	IF CommonTypesAndFunctions.StrEqualsAtStartWithDelimiter(str1:= ADR(LastTreeName), str2:= Data.PayloadString, delimiter:= SplitPayloadChar) THEN
		//now search split char
		StrPt := Data.PayloadString;
		StrPt := StrPt + TO_DWORD(CommonTypesAndFunctions.find(str1 := StrPt, str2:= ADR(SplitPayloadChar))) + 1;
		Target := StrPt^;
	END_IF
END_IF
END_METHOD

METHOD initAsFindTopic : BOOL
VAR_INPUT
END_VAR
getLastTreeName();
splitPayload := FALSE;
splitTopic := TRUE;
END_METHOD

METHOD getLastTreeName : BOOL
VAR_INPUT
END_VAR
LastTreeName := CommonTypesAndFunctions.FindLastDot(ADR(instanceName))^;
END_METHOD

METHOD initAsFindPayload : BOOL
VAR_INPUT
	//only first char is selected
	splitChar:STRING;
END_VAR
getLastTreeName();
splitPayload := TRUE;
splitTopic := FALSE;

SplitPayloadChar := CommonTypesAndFunctions.GetChar(in:= splitChar);
END_METHOD

END_FUNCTION_BLOCK

// MQTT/TestCases/Test Interfaces/exampleForFbs
FUNCTION_BLOCK exampleForFbs
VAR_INPUT
END_VAR
VAR_OUTPUT
END_VAR
VAR
	//the MQTT client
	//client:ClientWrapper;
	//some reciving FBs
	FirstExtReceiver:FooBarReceivingFB;
	SecondExtReceiver:FooBarReceivingFB;
	ThirdExtReceiver:FooBarReceivingFB;
	FourthExtReceiver:FooBarReceivingFB;
	//a Array of receiving FBs
	ArrayReceive:ARRAY[0..9] OF FooBarReceivingFB;
	
	//the collector of the FBs
	stock:CallbackCollector;
END_VAR



(*
client(
	broker:= 'test.mosquitto.org:1883', 
	connect:= TRUE, 
	tls:= FALSE);

	*)

END_FUNCTION_BLOCK

// MQTT/Function Blocks/CallbackFBs/Callback Collector/ReceiveValueWithStrucur
FUNCTION_BLOCK ReceiveValueWithStrucur EXTENDS ReceiveValue
VAR_INPUT
END_VAR
VAR_OUTPUT
END_VAR
VAR
	InstanceName:CommonTypesAndFunctions.GetInstanceName;
	localCompString:STRING(255);
END_VAR

METHOD InitReceiveStructur : BOOL
VAR_INPUT
	
	TopicLevel:USINT;
	//this typ is my received string
	ValueTyp:CommonTypesAndFunctions.VAR_TYPES; 
	//if set to true and hit we will return true, else false...
	returnHit: BOOL;
END_VAR
VAR
	tString:STRING(255);
	cmpByte:BYTE;
	bytePointer:POINTER TO BYTE;
	StringPointer:POINTER TO STRING;
	i:UINT;
END_VAR

tString:= InstanceName.GetInstanceTopic();

cmpByte:= CommonTypesAndFunctions.GetChar('/');

bytePointer := ADR(tString) + CommonTypesAndFunctions.len(ADR(tString));

i := 0;

WHILE bytePointer >= ADR(tString) DO
	IF bytePointer^ = cmpByte THEN
		i := i + 1; 
	END_IF
	
	IF i = TopicLevel THEN
		
		StringPointer := bytePointer + 1;
		//ReceiveTopic := GVL_ZIGBEE.TextZigbeeTopic;
		//ReceiveTopic := CONCAT(STR1:= ReceiveTopic, STR2:= StringPointer^); 
		localCompString := StringPointer^;
		initAsFindTopic(compString:= ADR(localCompString), ValueTyp:= ValueTyp, returnHit:= returnHit);
		RETURN;
	END_IF
	bytePointer := bytePointer - 1;
END_WHILE
localCompString := tString;
initAsFindTopic(compString:= ADR(localCompString), ValueTyp:= ValueTyp, returnHit:= returnHit);
END_METHOD

END_FUNCTION_BLOCK

// MQTT/Function Blocks/CallbackFBs/Callback Collector/ReceiveValue
(*
Receives one value from a MQTT publish packet.
It can check diffrent sources to determinate if the data is for this Value....

*)
FUNCTION_BLOCK ReceiveValue IMPLEMENTS MQTT_SUBSCRIBE_CALLBACK
VAR_INPUT
END_VAR
VAR_OUTPUT
	//your desired payload...
	MQTTReceived:CommonTypesAndFunctions.ALL_TYPES_UNION;
END_VAR
VAR
	//pointer to target
	TargetPointer:CommonTypesAndFunctions.ALL_TYPES_UNION_POINTER;
	//Target var type
	MyValueTyp:CommonTypesAndFunctions.VAR_TYPES;
	//an this is the split char...
	SplitPayloadChar: BYTE;
	//compare with this...
	MyCompString:POINTER TO STRING;
	//and this for Payload
	MyCompStringPayload:POINTER TO STRING;
	//if set to true and hit we will return true, else false...
	MyReturnHit: BOOL;
	ReceiveType : RECEIVE_TYPS;
END_VAR


METHOD PublishReceived : BOOL
VAR_INPUT
	(*Collection of received Data*)
	Data	: CALLBACK_DATA;
END_VAR
VAR
	StrPt : POINTER TO STRING;
END_VAR
CASE ReceiveType OF
	RECEIVE_TYPS.FIND_LAST_TOPIC:	
		//now search the right topic 
		IF CommonTypesAndFunctions.StrEquals(str1:= Data.TopicOutSplit^.Topics[Data.TopicOutSplit^.ValidFields - 1], str2:= MyCompString) THEN
			CommonTypesAndFunctions.GetValueFromStringPt(TypeOfValue:= MyValueTyp ,Target:= TargetPointer, str:= DATA.PayloadString);
			PublishReceived := MyReturnHit;
		END_IF
	RECEIVE_TYPS.FIND_PAYLOAD:
		IF CommonTypesAndFunctions.StrEqualsAtStartWithDelimiter(str1:= MyCompString, str2:= Data.PayloadString, delimiter:= SplitPayloadChar) THEN
			//now search split char
			StrPt := Data.PayloadString;
			StrPt := StrPt + TO_DWORD(CommonTypesAndFunctions.find(str1 := StrPt, str2:= ADR(SplitPayloadChar))) + 1;
			CommonTypesAndFunctions.GetValueFromStringPt(TypeOfValue:= MyValueTyp ,Target:= TargetPointer, str:= StrPt);
			PublishReceived := MyReturnHit;
		END_IF
	RECEIVE_TYPS.FIND_LAST_TOPIC_AND_PAYLOAD:
		//now search the right topic and payload
		IF CommonTypesAndFunctions.StrEquals(str1:= Data.TopicOut, str2:= MyCompString) THEN
			IF CommonTypesAndFunctions.StrEqualsAtStartWithDelimiter(str1:= MyCompStringPayload, str2:= Data.PayloadString, delimiter:= SplitPayloadChar) THEN
				StrPt := Data.PayloadString;
				StrPt := StrPt + TO_DWORD(CommonTypesAndFunctions.find(str1 := StrPt, str2:= ADR(SplitPayloadChar))) + 1;
				CommonTypesAndFunctions.GetValueFromStringPt(TypeOfValue:= MyValueTyp ,Target:= TargetPointer, str:= StrPt);
				PublishReceived := MyReturnHit;
			END_IF
		END_IF
	RECEIVE_TYPS.FIND_TOPIC:
		//now search the right topic 
		IF CommonTypesAndFunctions.StrEquals(str1:= Data.TopicOut, str2:= MyCompString) THEN
			CommonTypesAndFunctions.GetValueFromStringPt(TypeOfValue:= MyValueTyp ,Target:= TargetPointer, str:= DATA.PayloadString);
			PublishReceived := MyReturnHit;
		END_IF
END_CASE
END_METHOD

METHOD initAsFindPayload : BOOL
VAR_INPUT
	//only first char is selected
	splitChar:STRING;
	//this i'm searching
	compString : POINTER TO STRING;
	//this typ is my received string
	ValueTyp:CommonTypesAndFunctions.VAR_TYPES; 
	//if set to true and hit we will return true, else false...
	returnHit: BOOL;
END_VAR
ReceiveType := RECEIVE_TYPS.FIND_PAYLOAD;

SplitPayloadChar := CommonTypesAndFunctions.GetChar(in:= splitChar);
MyCompString := compString;
MyValueTyp := ValueTyp;
makePointer();
MyReturnHit := returnHit;
END_METHOD

(*this will only check the lowest topic level*)
METHOD initAsFindTopic : BOOL
VAR_INPUT
	//this i'm searching
	compString : POINTER TO STRING;
	//this typ is my received string
	ValueTyp:CommonTypesAndFunctions.VAR_TYPES; 
	//if set to true and hit we will return true, else false...
	returnHit: BOOL;
END_VAR
ReceiveType := RECEIVE_TYPS.FIND_TOPIC;
MyCompString := compString;
MyValueTyp := ValueTyp;
makePointer();
MyReturnHit := returnHit;
END_METHOD

METHOD makePointer : BOOL
VAR_INPUT
END_VAR
TargetPointer := CommonTypesAndFunctions.MakeAllTypesPointer(fromWho:= adr(MQTTReceived), myType:= MyValueTyp);
END_METHOD

(*this will check the whole topic!*)
METHOD initAsFindTopicAndPayload : BOOL
VAR_INPUT
	//only first char is selected
	splitChar:STRING;
	//this topic i'm searching
	compStringTopic : POINTER TO STRING;
	//this payload i'm searching
	compStringPayload : POINTER TO STRING;
	//this typ is my received string
	ValueTyp:CommonTypesAndFunctions.VAR_TYPES; 
	//if set to true and hit we will return true, else false...
	returnHit: BOOL;
END_VAR
ReceiveType := RECEIVE_TYPS.FIND_LAST_TOPIC_AND_PAYLOAD;
SplitPayloadChar := CommonTypesAndFunctions.GetChar(in:= splitChar);
MyCompString := compStringTopic;
MyCompStringPayload := compStringPayload;
MyValueTyp := ValueTyp;
makePointer();
MyReturnHit := returnHit;
END_METHOD

METHOD SetOutput : BOOL
VAR_INPUT
	value:CommonTypesAndFunctions.ALL_TYPES_UNION;
END_VAR
MQTTReceived := value;
END_METHOD

METHOD initAsFindLastTopic : BOOL
VAR_INPUT
	//this i'm searching
	compString : POINTER TO STRING;
	//this typ is my received string
	ValueTyp:CommonTypesAndFunctions.VAR_TYPES; 
	//if set to true and hit we will return true, else false...
	returnHit: BOOL;
END_VAR
ReceiveType := RECEIVE_TYPS.FIND_LAST_TOPIC;
MyCompString := compString;
MyValueTyp := ValueTyp;
makePointer();
MyReturnHit := returnHit;
END_METHOD

END_FUNCTION_BLOCK

// MQTT/Function Blocks/CallbackFBs/Callback Collector/ReceiveString
FUNCTION_BLOCK ReceiveString IMPLEMENTS MQTT_SUBSCRIBE_CALLBACK
VAR_INPUT
END_VAR
VAR_OUTPUT
	//your desired payload...
	MQTTReceived:STRING(255);
END_VAR
VAR
	//if set to true we search the instance name in the lowest topic
	splitTopic: BOOL;
	//if set to true we search the instance name in Payload separatet by the split char 
	splitPayload: BOOL;
	//an this is the split char...
	SplitPayloadChar: BYTE;
	//compare with this...
	MyCompString:POINTER TO STRING;
	//if set to true and hit we will return true, else false...
	MyReturnHit: BOOL;
END_VAR

METHOD PublishReceived : BOOL
VAR_INPUT
	(*Collection of received Data*)
	Data	: CALLBACK_DATA;
	
END_VAR
VAR
	StrPt : POINTER TO STRING(255);
END_VAR
// no we can check if the topic/payload matches to my compare string 

//now search the right topic 
IF splitTopic THEN
	
	IF CommonTypesAndFunctions.StrEquals(str1:= Data.TopicOut, str2:= MyCompString) THEN
		StrPt := Data.PayloadString;
		MQTTReceived := StrPt^;
		PublishReceived := MyReturnHit;
	END_IF

END_IF

//now look into the payload
IF splitPayload THEN
	
	IF CommonTypesAndFunctions.StrEqualsAtStartWithDelimiter(str1:= MyCompString, str2:= Data.PayloadString, delimiter:= SplitPayloadChar) THEN
		//now search split char
		StrPt := Data.PayloadString;
		StrPt := StrPt + TO_DWORD(CommonTypesAndFunctions.find(str1 := StrPt, str2:= ADR(SplitPayloadChar))) + 1;
		MQTTReceived := StrPt^;
		PublishReceived := MyReturnHit;
	END_IF
END_IF
END_METHOD

METHOD initAsFindTopic : BOOL
VAR_INPUT
	//this i'm searching
	compString : POINTER TO STRING;
	//if set to true and hit we will return true, else false...
	returnHit: BOOL;
END_VAR

splitPayload := FALSE;
splitTopic := TRUE;
MyCompString := compString;
MyReturnHit := returnHit;
END_METHOD

METHOD initAsFindPayload : BOOL
VAR_INPUT
	//only first char is selected
	splitChar:STRING;
	//this i'm searching
	compString : POINTER TO STRING;
	//if set to true and hit we will return true, else false...
	returnHit: BOOL;
END_VAR

splitPayload := TRUE;
splitTopic := FALSE;

SplitPayloadChar := CommonTypesAndFunctions.GetChar(in:= splitChar);
MyCompString := compString;
MyReturnHit := returnHit;
END_METHOD

END_FUNCTION_BLOCK

// MQTT/TestCases/TestLongPublish
FUNCTION_BLOCK TestLongPublish
VAR_INPUT
	broker:STRING := 'test.mosquitto.org:1883';
END_VAR
VAR_OUTPUT
END_VAR
VAR
	longPayload:STRING(8000):='';
	longTopic:STRING(8000):=('TestTopic/');
	longPayloadReceive:STRING(8000);
	longTopicReceive:STRING(8000);
	init: BOOL;
	i1:UINT;
	i2:UINT;
	countAsciis :UINT := 48;
	pt1:POINTER TO BYTE;
	pt2:POINTER TO BYTE;
	
	step : UINT; 
	
	MQTT:HANDLE_MQTT;
	
	MQTT_IN_OUT:MQTT_IN_OUT;
	
	ComConfig:COM_CONFIG;
	
	pup:MQTTPublish;
	send: BOOL;

	
	SUB1:MQTTSubscribe;
	subscribe: BOOL;

	callback : SingelStringCallback;
	
	
	connect: BOOL;

	nextRung:ton;
	lenPayload:UINT;
	lenTopic:uint;
	
END_VAR

IF NOT init THEN
	init := TRUE;
	SUB1.SetMqttInOut(MQTT_IN_OUT := ADR(MQTT_IN_OUT));
	pup.SetMqttInOut(MQTT_IN_OUT := ADR(MQTT_IN_OUT));
	ComConfig.MaxPayloadSize := 20000;
	ComConfig.MaxTopicLevels := 10;
	ComConfig.MaxTopicElementSize := 10000;
	
	MQTT_IN_OUT.ClientID := 'TestCodesys';
	MQTT_IN_OUT.COM_CONFIG := ComConfig;
	//firs build some nice pacload ...
	pt1 := ADR(longPayload);
	pt2 := ADR(longTopic);
	pt2 := pt2 + 10;
	FOR i1 := 0 TO 8000 / countAsciis - 1 DO
		FOR i2 := 0 TO countAsciis - 1 DO
			pt1^ := TO_BYTE(i2 + 16#30); //16#30 --> ASCII zero
			pt2^ := TO_BYTE(i2 + 16#30); //16#30 --> ASCII zero
			pt1 := pt1 + 1;
			pt2 := pt2 + 1;
		END_FOR
	END_FOR
	//need termination...
	pt1^:= 0;
	pt2^:= 0;
	callback.Init(payload:= ADR(longPayloadReceive), topic:= ADR(longTopicReceive));
END_IF

SUB1(
	Subscribe:= subscribe, 
	Topic:= ADR('TestTopic/#'), 
	QoSSubscribe:= QoS.ExactlyOnce, 
	ExpectingString:= TRUE, 
	Callback:= callback);

	
	pup(
	Topic:= ADR(longTopic), 
	PayloadString:= ADR(longPayload), 
	PublishAsString:= TRUE, 
	QoSIn:= Qos.ExactlyOnce, 
	MRetain:= FALSE, 
	send:= send);

MQTT(
	MQTT_IN_OUT:= MQTT_IN_OUT, 
	ENABLE:= connect, 
	URL:= broker, 
	TIMEOUT:= T#5S);


CASE step OF 
	0://begin
		//connect
		connect := TRUE;
		step := 10;
	10://wait connected
		IF MQTT_IN_OUT.BROKER_CONNECTED THEN
			//subscribe
			subscribe := TRUE;		
			step := 20;
		END_IF
	20://wait subscribed
		IF SUB1.SubscribeDone THEN
			//send packet and check receive
			send := TRUE;
			step := 30;
		END_IF
		
	30:
		//reset send
		send := FALSE;
		step := 40;
	40:
		lenPayload:= CommonTypesAndFunctions.len(ADR(longPayloadReceive));
		lenTopic:= CommonTypesAndFunctions.len(ADR(longTopicReceive));
		//check if payload and topic received....
		IF CommonTypesAndFunctions.StrEquals(str1:= ADR(longPayload), str2:= ADR(longPayloadReceive)) AND
			CommonTypesAndFunctions.StrEquals(str1:= ADR(longTopic), str2:= ADR(longTopicReceive)) THEN
			//deled received strings
			longTopicReceive := '';
			longPayloadReceive := '';
			//go wait repeat
			step := 50;
		END_IF
		
	50:
		IF nextRung.Q THEN
			step := 0;
		END_IF
END_CASE

nextRung(IN:= step = 50, PT:= T#5S);

END_FUNCTION_BLOCK

// MQTT/TestCases/TestLongStringList
FUNCTION_BLOCK TestLongStringList
VAR_INPUT
	//use this input if you want to test with another broker
	client:STRING:='test.mosquitto.org:1883';//test.mosquitto.org
	
END_VAR
VAR_OUTPUT
END_VAR
VAR
	MQTTClient:HANDLE_MQTT;
	MQTT_IN_OUT:MQTT_IN_OUT;
	MQTTInfo:MQTT_INFO;
	publish:MQTTPublish;
	subscribe:MQTTSubscribe;
	ReceiveSubscribeTopic:STRING(255);
	
	ReceiveSubscribePayloadLong:STRING(500);
	State :MQTTState;
	init: BOOL;
	varSend: BOOL;
	timerSend:ton;
	t1:ton;
	t2:ton;
	Payload:STRING;
	//the method PublishReceved() is call when an publsih packet form the broker is received.
	StringCallback:ListStringCallback;
	//the array contains the targets and sub topics for receive
	CallBackTargets:ARRAY[0..1] OF LIST_STRING_CALLBACK_DATA := [(Target:=ADR(ReceiveSubscribePayloadLong), SubTopic:= ADR('Long'))];
	len1:UINT;
END_VAR

//here init is done
IF NOT init THEN
	init := TRUE;
	MQTT_IN_OUT.ClientID := CONCAT('CodesysMqtt',TO_STRING(TICKS.GetTick(xDummy:= TRUE)));
	//init state FB, so you only have to call state();without parameters... 
	State.Init(
	State:= ADR(t1.Q), 
	Topic:= ADR('CODESYS-MQTT-BY-SD/Long'), 
	StateName:= ADR(''), 
	StateValueOn:= ADR('LOOOOOOOOOOOOOOOOOOOOOOOOOOOOOOOOOOOOOOOOOOOOOOOOOOOOOOOOOOOOOOOOOOOOOOOOOOOOOOOOOOOOOOOOOOOOOOOOOOOOOOOOOOOOOOOOOOOOOOOOOOOOOOOOOOOOOOOOOOOOOOOOOOOOOOOOOOOOOOOOOOOOOOOOOOOOOOOOOOOOOOOOOOOOOOOOOOOOOOOOOOOOOOOOOOOOOOOOg:On'), 
	StateValueOff:= ADR('LOOOOOOOOOOOOOOOOOOOOOOOOOOOOOOOOOOOOOOOOOOOOOOOOOOOOOOOOOOOOOOOOOOOOOOOOOOOOOOOOOOOOOOOOOOOOOOOOOOOOOOOOOOOOOOOOOOOOOOOOOOOOOOOOOOOOOOOOOOOOOOOOOOOOOOOOOOOOOOOOOOOOOOOOOOOOOOOOOOOOOOOOOOOOOOOOOOOOOOOOOOOOOOOOOOOOOOOOg:Off'), 
	QoS:= QoS.ExactlyOnce, 
	RetainMqtt:= TRUE,
	MQTT_IN_OUT:= ADR(MQTT_IN_OUT));
	StringCallback.InitAsSplitTopic(ListData := ADR(CallBackTargets), LengthOfData:= 1);
	
	subscribe.SetMqttInOut(MQTT_IN_OUT:= ADR(MQTT_IN_OUT));
	
END_IF
//timer for repeating packets
t1(IN:= NOT t2.Q, PT:= T#1S, );
t2(IN:= t1.Q, PT:= T#1S);
//call of MQTT client
MQTTClient(
	MQTT_IN_OUT:= MQTT_IN_OUT, 
	ENABLE:= TRUE, 
	URL:= client, 
	TIMEOUT:= T#5S, 
	TLS:= FALSE);
//Subscribe to topic
subscribe(
	Subscribe:= TRUE, 
	Topic:= ADR('CODESYS-MQTT-BY-SD/#'), 
	QoSSubscribe:= QoS.ExactlyOnce, 
	ExpectingString:= TRUE,
	Callback:= StringCallback);
len1 := CommonTypesAndFunctions.len(str:= ADR(ReceiveSubscribePayloadLong));

//call of state FB
State();

END_FUNCTION_BLOCK

// MQTT/TestCases/TestStringPointer
FUNCTION_BLOCK TestStringPointer
VAR_INPUT
END_VAR
VAR_OUTPUT
END_VAR
VAR
	SFrom:STRING(2000):='ABCDEFGHIJKLMNOPQRSTUVWXYZABCDEFGHIJKLMNOPQRSTUVWXYZABCDEFGHIJKLMNOPQRSTUVWXYZABCDEFGHIJKLMNOPQRSTUVWXYZABCDEFGHIJKLMNOPQRSTUVWXYZABCDEFGHIJKLMNOPQRSTUVWXYZABCDEFGHIJKLMNOPQRSTUVWXYZABCDEFGHIJKLMNOPQRSTUVWXYZABCDEFGHIJKLMNOPQRSTUVWXYZABCDEFGHIJKLMNOPQRSTUVWXYZABCDEFGHIJKLMNOPQRSTUVWXYZABCDEFGHIJKLMNOPQRSTUVWXYZABCDEFGHIJKLMNOPQRSTUVWXYZABCDEFGHIJKLMNOPQRSTUVWXYZABCDEFGHIJKLMNOPQRSTUVWXYZABCDEFGHIJKLMNOPQRSTUVWXYZABCDEFGHIJKLMNOPQRSTUVWXYZABCDEFGHIJKLMNOPQRSTUVWXYZABCDEFGHIJKLMNOPQRSTUVWXYZABCDEFGHIJKLMNOPQRSTUVWXYZABCDEFGHIJKLMNOPQRSTUVWXYZABCDEFGHIJKLMNOPQRSTUVWXYZABCDEFGHIJKLMNOPQRSTUVWXYZABCDEFGHIJKLMNOPQRSTUVWXYZABCDEFGHIJKLMNOPQRSTUVWXYZABCDEFGHIJKLMNOPQRSTUVWXYZABCDEFGHIJKLMNOPQRSTUVWXYZABCDEFGHIJKLMNOPQRSTUVWXYZABCDEFGHIJKLMNOPQRSTUVWXYZABCDEFGHIJKLMNOPQRSTUVWXYZABCDEFGHIJKLMNOPQRSTUVWXYZABCDEFGHIJKLMNOPQRSTUVWXYZABCDEFGHIJKLMNOPQRSTUVWXYZABCDEFGHIJKLMNOPQRSTUVWXYZABCDEFGHIJKLMNOPQRSTUVWXYZABCDEFGHIJKLMNOPQRSTUVWXYZABCDEFGHIJKLMNOPQRSTUVWXYZABCDEFGHIJKLMNOPQRSTUVWXYZABCDEFGHIJKLMNOPQRSTUVWXYZABCDEFGHIJKLMNOPQRSTUVWXYZABCDEFGHIJKLMNOPQRSTUVWXYZABCDEFGHIJKLMNOPQRSTUVWXYZABCDEFGHIJKLMNOPQRSTUVWXYZABCDEFGHIJKLMNOPQRSTUVWXYZABCDEFGHIJKLMNOPQRSTUVWXYZABCDEFGHIJKLMNOPQRSTUVWXYZABCDEFGHIJKLMNOPQRSTUVWXYZABCDEFGHIJKLMNOPQRSTUVWXYZABCDEFGHIJKLMNOPQRSTUVWXYZABCDEFGHIJKLMNOPQRSTUVWXYZABCDEFGHIJKLMNOPQRSTUVWXYZABCDEFGHIJKLMNOPQRSTUVWXYZABCDEFGHIJKLMNOPQRSTUVWXYZABCDEFGHIJKLMNOPQRSTUVWXYZABCDEFGHIJKLMNOPQRSTUVWXYZABCDEFGHIJKLMNOPQRSTUVWXYZABCDEFGHIJKLMNOPQRSTUVWXYZABCDEFGHIJKLMNOPQRSTUVWXYZABCDEFGHIJKLMNOPQRSTUVWXYZABCDEFGHIJKLMNOPQRSTUVWXYZABCDEFGHIJKLMNOPQRSTUVWXYZABCDEFGHIJKLMNOPQRSTUVWXYZABCDEFGHIJKLMNOPQRSTUVWXYZABCDEFGHIJKLMNOPQRSTUVWXYZABCDEFGHIJKLMNOPQRSTUVWXYZABCDEFGHIJKLMNOPQRSTUVWXYZABCDEFGHIJKLMNOPQRSTUVWXYZABCDEFGHIJKLMNOPQRSTUVWXYZ';
	STo:STRING(1000):='';
	p1:POINTER TO STRING(2000);
	p2:POINTER TO STRING(2000);
	l1:UINT;
	l2:UINT;
END_VAR

l1 := CommonTypesAndFunctions.len(str:= ADR(SFrom));
l2 := CommonTypesAndFunctions.len(str:= ADR(STo));
p1:= ADR(SFrom);
p2:= ADR(STo);
p2^:= p1^;

END_FUNCTION_BLOCK

// MQTT/TestCases/TestUserPassword
FUNCTION_BLOCK TestUserPassword
VAR_INPUT
END_VAR
VAR_OUTPUT
END_VAR
VAR
MQTT1:HANDLE_MQTT ;
MQTT2:HANDLE_MQTT ;
MQTT3:HANDLE_MQTT ;	
info:MQTT_INFO;
MQTT_IN_OUT:MQTT_IN_OUT;
END_VAR

MQTT1(MQTT_IN_OUT := MQTT_IN_OUT,
	ENABLE := TRUE,
	URL:= 'User1:Mypassword@test.mosquitto.org:1883');
	
MQTT2(MQTT_IN_OUT := MQTT_IN_OUT,
	ENABLE := TRUE,
	URL:= 'User1@test.mosquitto.org:1883');
	
MQTT3(MQTT_IN_OUT := MQTT_IN_OUT,
	ENABLE := TRUE,
	URL:= 'User2:Mypassword@test.mosquitto.org:1883');

END_FUNCTION_BLOCK

// MQTT/Function Blocks/CallbackFBs/Callback Collector/ReceiverBase
FUNCTION_BLOCK ReceiverBase
VAR_INPUT
END_VAR
VAR_OUTPUT
END_VAR
VAR
	MatchTyp:RECEIVER_INIT_TYPS;
	Target:CommonTypesAndFunctions.ALL_TYPES_UNION_POINTER;
	TargetType:CommonTypesAndFunctions.VAR_TYPES;
	PayloadCompare:POINTER TO STRING;
	TopicCompare:POINTER TO STRING;
	delimiter:BYTE;
	delimiterString:STRING(3);
	SplitTopic:HandleSplitTopic;
END_VAR

METHOD init
VAR_INPUT
	MQTT_IN_OUT:POINTER TO MQTT_IN_OUT;
	MatchTyp:RECEIVER_INIT_TYPS;
	Target:CommonTypesAndFunctions.ALL_TYPES_UNION_POINTER;
	TargetType:CommonTypesAndFunctions.VAR_TYPES;
	PayloadCompare:POINTER TO STRING;
	TopicCompare:POINTER TO STRING;
	delimiter:BYTE;
	
END_VAR
MatchTyp := MatchTyp;
Target := Target;
TargetType := TargetType;
PayloadCompare := PayloadCompare;
TopicCompare := TopicCompare;
delimiter := delimiter;
delimiterString[0] := delimiter;
delimiterString[1] := 0;

IF MatchTyp = RECEIVER_INIT_TYPS.MQTT_STRING or MatchTyp = RECEIVER_INIT_TYPS.MQTT_STRING_JSON THEN
	SplitTopic.LowInit(TopicsLevelInit:= MQTT_IN_OUT^.COM_CONFIG.MaxTopicLevels,
			 SplitElementSizeInit:= MQTT_IN_OUT^.COM_CONFIG.MaxTopicElementSize, dynMemUsageInit:= ADR(MQTT_IN_OUT^.dynMemUsage));
	SplitTopic.NewTopic(in:= TopicCompare, test:= TRUE, SizeOfString:= CommonTypesAndFunctions.len(str:= TopicCompare));
END_IF
END_METHOD

METHOD CheckMatch : BOOL
VAR_INPUT
	(*Collection of received Data*)
	Data	: CALLBACK_DATA;
END_VAR
VAR 
	foundPos:DINT;
END_VAR
CheckMatch := FALSE;
CASE MatchTyp OF
	RECEIVER_INIT_TYPS.FIND_FULL_TOPIC:
		IF CommonTypesAndFunctions.StrEquals(str1:= Data.TopicOut , str2:= PayloadCompare) THEN
			CheckMatch := TRUE;
			GetValue(fromWhere:= Data.PayloadString);
			RETURN;
		END_IF 
	RECEIVER_INIT_TYPS.FIND_LAST_TOPIC:
		IF CommonTypesAndFunctions.StrEquals(str1:= Data.TopicOutSplit^.Topics[Data.TopicOutSplit^.ValidFields - 1], str2:= PayloadCompare) THEN
			CheckMatch := TRUE;
			GetValue(fromWhere:= Data.PayloadString);
			RETURN;
		END_IF
	RECEIVER_INIT_TYPS.FIND_PAYLOAD:
		IF CommonTypesAndFunctions.StrEqualsAtStartWithDelimiter(str1:= PayloadCompare, str2:= Data.PayloadString , delimiter:= delimiter) THEN
			CheckMatch := TRUE;
			GetValue(fromWhere:= Data.PayloadString + TO_UINT(CommonTypesAndFunctions.find(str1:= Data.PayloadString, str2:= ADR(delimiterString)))+1);
			RETURN;	
		END_IF
	RECEIVER_INIT_TYPS.JSON_FULL:
		IF CommonTypesAndFunctions.StrEquals(str1:= Data.TopicOut , str2:= PayloadCompare) THEN
			foundPos := CommonTypesAndFunctions.find(str1:= Data.PayloadString, str2:= TopicCompare); 
			IF foundPos >= 0 THEN
				CheckMatch := TRUE;
				RETURN;	
			END_IF
		END_IF
	RECEIVER_INIT_TYPS.JSON_SMALL:
		IF CommonTypesAndFunctions.StrEquals(str1:= Data.TopicOutSplit^.Topics[Data.TopicOutSplit^.ValidFields - 1], str2:= PayloadCompare) THEN
			IF CommonTypesAndFunctions.find(str1:= Data.PayloadString, str2:= TopicCompare) >= 0 THEN
				CheckMatch := TRUE;
				RETURN;	
			END_IF
		END_IF
	RECEIVER_INIT_TYPS.MQTT_STRING:
		IF SplitTopic.CheckTopicMatchToMe(with:= Data.TopicOutSplit) = TOPIC_MATCH.TOPIC_MATCHES THEN
			CheckMatch := TRUE;
			RETURN;
		END_IF
	RECEIVER_INIT_TYPS.MQTT_STRING_JSON:
		IF SplitTopic.CheckTopicMatchToMe(with:= Data.TopicOutSplit) = TOPIC_MATCH.TOPIC_MATCHES THEN
			IF CommonTypesAndFunctions.find(str1:= Data.PayloadString, str2:= TopicCompare) >= 0 THEN
				CheckMatch := TRUE;
				RETURN;	
			END_IF
		END_IF
	
END_CASE
END_METHOD

METHOD GetValue
VAR_INPUT
	fromWhere: POINTER TO STRING(65000);
END_VAR
CASE TargetType OF
	CommonTypesAndFunctions.VAR_TYPES.BOOL_T,
	CommonTypesAndFunctions.VAR_TYPES.BYTE_T,
	CommonTypesAndFunctions.VAR_TYPES.DATE_T,
	CommonTypesAndFunctions.VAR_TYPES.DINT_T,
	CommonTypesAndFunctions.VAR_TYPES.DT_T,
	CommonTypesAndFunctions.VAR_TYPES.DWORD_T,
	CommonTypesAndFunctions.VAR_TYPES.INT_T,
	CommonTypesAndFunctions.VAR_TYPES.LINT_T,
	CommonTypesAndFunctions.VAR_TYPES.LREAL_T,
	CommonTypesAndFunctions.VAR_TYPES.LWORD_T,
	CommonTypesAndFunctions.VAR_TYPES.REAL_T,
	CommonTypesAndFunctions.VAR_TYPES.SINT_T,
	CommonTypesAndFunctions.VAR_TYPES.TIME_T,
	CommonTypesAndFunctions.VAR_TYPES.TOD_T,
	CommonTypesAndFunctions.VAR_TYPES.TOD2_T,
	CommonTypesAndFunctions.VAR_TYPES.UDINT_T,
	CommonTypesAndFunctions.VAR_TYPES.UINT_T,
	CommonTypesAndFunctions.VAR_TYPES.ULINT_T,
	CommonTypesAndFunctions.VAR_TYPES.USINT_T,
	CommonTypesAndFunctions.VAR_TYPES.WORD_T:
	CommonTypesAndFunctions.GetValueFromStringPt
				(TypeOfValue:= TargetType, Target:= Target, str:= fromWhere);
END_CASE
END_METHOD

END_FUNCTION_BLOCK

// MQTT/TestCases/Test Interfaces/TestCallbackCollecktor
FUNCTION_BLOCK TestCallbackCollecktor
VAR_INPUT
END_VAR
VAR_OUTPUT
END_VAR
VAR
	var1:AllValuesCallback;
	var2:AllValuesCallback;
	var3:AllValuesCallback;
	collector:CallbackCollector;
	init: BOOL;
	target1:INT;
	pt1:CommonTypesAndFunctions.ALL_TYPES_UNION_POINTER;
	callbackData:CALLBACK_DATA;
	stringPayload:STRING :='123';
END_VAR

IF NOT init THEN
	init := TRUE;
	pt1.POINTER_TO_INT_T := ADR(target1);
	var1.Init(SetType := CommonTypesAndFunctions.VAR_TYPES.INT_T, Target := pt1);
	callbackData.PayloadString := ADR(stringPayload);
END_IF

//try delet without registert instance
collector.destroy();
//put one instance
collector.put(instance:= var1);

collector.PublishReceived(Data:= callbackData);

collector.destroy();

//put two instance
collector.put(instance:= var1);
collector.put(instance:= var1);

collector.PublishReceived(Data:= callbackData);

collector.destroy();

//put tree instance
collector.put(instance:= var1);
collector.put(instance:= var1);
collector.put(instance:= var1);

collector.PublishReceived(Data:= callbackData);

collector.destroy();

//put tree instance
collector.put(instance:= var1);
collector.put(instance:= var2);
collector.put(instance:= var3);

METHOD FB_Exit
VAR_INPUT 
 bInCopyCode : BOOL; // TRUE: the exit method is called in order to leave the instance which will be copied afterwards (online change). 
END_VAR
collector.destroy();
END_METHOD

END_FUNCTION_BLOCK

// MQTT/TestCases/TestMemHandle
FUNCTION_BLOCK TestMemHandle
VAR_INPUT
END_VAR
VAR_OUTPUT
END_VAR
VAR
	MQTT_IN_OUT_1:MQTT_IN_OUT;
	MQTT_IN_OUT_2:MQTT_IN_OUT;
	Client1:HANDLE_MQTT;
	Client2:HANDLE_MQTT;
END_VAR

Client1(
	MQTT_IN_OUT:= MQTT_IN_OUT_1, 
	ENABLE:= TRUE, 
	URL:= 'test.mosquitto.org:1883', 
	TIMEOUT:= T#5S);
	
Client2(
	MQTT_IN_OUT:= MQTT_IN_OUT_2, 
	ENABLE:= TRUE, 
	URL:= 'test.mosquitto.org:1883', 
	TIMEOUT:= T#5S);

END_FUNCTION_BLOCK

// MQTT/TestCases/TestSplitTopic
FUNCTION_BLOCK TestSplitTopic
VAR_INPUT
END_VAR
VAR_OUTPUT
END_VAR
VAR
	Split1:HandleSplitTopic;
	Split2:HandleSplitTopic;
	Usage1:UDINT;
	Usage2:UDINT;
	COM_CONFIG:COM_CONFIG;
END_VAR

Split1.FullInit(TopicsLevelInit:= COM_CONFIG.MaxTopicLevels, SplitElementSizeInit:= COM_CONFIG.MaxTopicElementSize, dynMemUsageInit:= ADR(Usage1));
Split2.LowInit(TopicsLevelInit:= COM_CONFIG.MaxTopicLevels, SplitElementSizeInit:= COM_CONFIG.MaxTopicElementSize, dynMemUsageInit:= ADR(Usage1));

Split1.destroy();
Split2.destroy();

END_FUNCTION_BLOCK
